(* PLC project Unnamed, Unknown Unnamed 1 *)
(* stored: creationDateTime 2023-12-01T09:13:18, modificationDateTime 2023-12-01T09:35:23 *)

PROGRAM project_un
  VAR
    PB1 AT %IX0.0 : BOOL;
    PB2 AT %IX0.1 : BOOL;
    LED AT %QX0.0 : BOOL;
  END_VAR

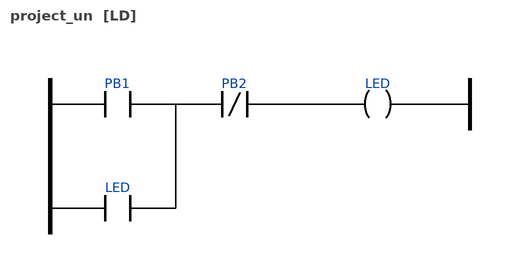
(* LD diagram, written out as Structured Text *)
LED := (PB1 OR LED) AND NOT PB2;
END_PROGRAM

CONFIGURATION Config0
  RESOURCE Res0 ON PLC
    VAR_GLOBAL
      PB1 AT %IX0.0 : BOOL;
      LAMP AT %QX0.0 : BOOL;
      PB2 AT %IX0.1 : BOOL;
    END_VAR
    TASK task0(INTERVAL := T#20ms, PRIORITY := 0);
    PROGRAM instance0 WITH task0 : project_un;
  END_RESOURCE
END_CONFIGURATION
